FUNCTION FUN_Add : REAL
VAR_INPUT
		f_Inp1			: REAL;
		f_Inp2			: REAL;
END_VAR
VAR
END_VAR

FUN_Add := f_Inp1 + f_Inp2;

END_FUNCTION

(* stored: Version 1.1.0.1, ProductVersion 3.1.4024.9
   POU FUN_Add: Id {da39f6b9-865b-4010-9a48-451276c105d7}, SpecialFunc None *)
